// TwinCAT 3 PLC project FirstPLC
// Title: TwinCAT_DSA
// Company: UBC
// ProjectVersion: 0.0.1
// ProgramVersion: 3.1.4026.10
// libraries:
//   Tc2_ControllerToolbox, * (Beckhoff Automation GmbH)
//   Tc2_MC2, * (Beckhoff Automation GmbH)
//   Tc2_Standard, * (Beckhoff Automation GmbH)
//   Tc2_System, * (Beckhoff Automation GmbH)
//   Tc2_Utilities, * (Beckhoff Automation GmbH)
//   Tc3_Module, * (Beckhoff Automation GmbH)
//   TwinCAT_DSA, * (UBC)
// project tree:
//   / PlcTask.TcTTO
//   POUs/ MAIN.TcPOU, SimplePID.TcPOU
// real-time tasks:
//   TASK PlcTask: cycle T#1ms, priority 20, ADS port 350
//   TASK PlcTask1: cycle T#1ms, priority 21, ADS port 351
// motion (NC):
//   TASK NC-Task 1 SAF: cycle T#1ms, priority 4, ADS port 501
//   TASK NC-Task 1 SVB: cycle T#10ms, priority 8, ADS port 511
//   AXIS Axis 1 (id 1)
//     OtherSettings: AllowMotionCmdToSlave=true
//     encoder EncType=1
//     drive DrvType=5
//       Analog: TorqueSetpointScale=10, ScaleFactorActTorque=0.1
//       TimeComp: TaskDelayCycles=1
//     controller CtrType=1
//       CtrPara: PriorControlFactor=1
//         Observer: BandWidth=20
// variable links:
//   FirstPLC/FirstPLC Instance <-> PlantSimulator/PlantSimulator Instance
//     PlcTask Inputs/MAIN.lrActualPosition <-> PlcTask Outputs/MAIN.lrOutput
//     PlcTask Outputs/MAIN.lrControllerOutput <-> PlcTask Inputs/MAIN.lrIn

CONFIGURATION FirstPLC
    RESOURCE PLC ON TwinCAT3
        TASK PlcTask(INTERVAL := T#1ms, PRIORITY := 20);
        PROGRAM MAIN WITH PlcTask : MAIN;
    END_RESOURCE
END_CONFIGURATION

// ---- POUs/MAIN.TcPOU
PROGRAM MAIN
VAR
    nState : INT := 0;
    fbMyPid : SimplePID;
    lrKp : LREAL := 1000.000;
    lrTn : LREAL := 0.159200;
    lrTv : LREAL := 0.0031847;
    lrTd : LREAL := 0.07647;
    lrActualPosition AT%I* : LREAL;
    lrControllerOutput AT%Q* : LREAL;
    lrSetpoint : LREAL := 0.0;
END_VAR

CASE nState OF
    10:
        fbMyPid.lrKp := lrKp;
        fbMyPid.lrTn := lrTn;
        fbMyPid.lrTv := lrTv;
        fbMyPid.lrTd := lrTd;

        fbMyPid(
            lrSetpointPosition := lrSetpoint,
            lrActualPosition := lrActualPosition,
            bStart := TRUE,
            lrControlOutput => lrControllerOutput
        );
END_CASE

END_PROGRAM

// ---- POUs/SimplePID.TcPOU
FUNCTION_BLOCK SimplePID
VAR_INPUT
	lrActualPosition : LREAL := 0.0;
	lrSetpointPosition : LREAL := 0.0;
	lrKp : LREAL := 1.0;
	lrTn :LREAL := 1.0;
	lrTv : LREAL := 0.0;
	lrTd : LREAL := 0.0;
	bStart : BOOL := FALSE;
END_VAR

VAR_OUTPUT
	lrControlOutput : LREAL :=0.0;
END_VAR

VAR
	lrTs : LREAL := 0.001; //1ms
	nState : INT := 0;	
	lrError : LREAL := 0.0;
	lrD : LREAL := 0.0;
	lrKi : Lreal := 0.0;
	lrKd: LREAL := 0.0;
	lrK1: LREAL := 0.0;
	lrP: LREAL := 0.0;
	lrI: LREAL := 0.0;
	lrLastI: LREAL := 0.0;
	lrLastError: LREAL := 0.0;
	lrLastD: LREAL := 0.0;
	
	MAX_INTEGRAL: LREAL := 1;
	MIN_INTEGRAL: LREAL := -1;
END_VAR

CASE nState OF 
	0:
		IF bStart THEN
			nState := 10;
		END_IF
	
	10:
		IF bStart = FALSE THEN
			nState := 0;	
		END_IF
		
		lrError := lrSetpointPosition - lrActualPosition;
		lrKi := lrKp * lrTs / lrTn;
		lrKd := lrKp * lrTv / (lrTd + lrTs);
		lrK1 := lrTd / (lrTd + lrTs);
		lrP := lrKp * lrError;
		lrI := lrLastI + lrKi * lrError; 
		lrD := lrK1 * lrLastD + lrKd * (lrError - lrLastError);
		lrControlOutput := lrP + lrI + lrD;
		
		//Integrator wind up
		
		IF lrI > MAX_INTEGRAL THEN
			lrI := MAX_INTEGRAL;
		ELSIF lrI < MIN_INTEGRAL THEN
			lrI := MIN_INTEGRAL;
		END_IF
		
		lrLastError := lrError;
		lrLastD := lrD;
		lrLastI := lrI;
END_CASE

END_FUNCTION_BLOCK
